FUNCTION_BLOCK POSTGRE_DB_INSERT
  {SET_ATTRIBUTE(OpcUa, POINT.ENDPOINT)}
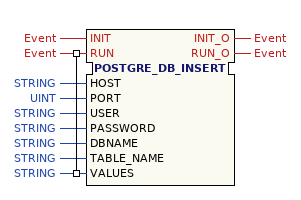
  EVENT_INPUT
    INIT;
    RUN WITH VALUES;
  END_EVENT
  EVENT_OUTPUT
    INIT_O;
    RUN_O;
  END_EVENT
  VAR_INPUT
    HOST : STRING; {SET_ATTRIBUTE(OpcUa, Constant)}
    PORT : UINT; {SET_ATTRIBUTE(OpcUa, Constant)}
    USER : STRING; {SET_ATTRIBUTE(OpcUa, Constant)}
    PASSWORD : STRING; {SET_ATTRIBUTE(OpcUa, Constant)}
    DBNAME : STRING; {SET_ATTRIBUTE(OpcUa, Constant)}
    TABLE_NAME : STRING; {SET_ATTRIBUTE(OpcUa, Constant)}
    VALUES : STRING; {SET_ATTRIBUTE(OpcUa, Constant)}
  END_VAR
END_FUNCTION_BLOCK
